TYPE ST_EL3446_MUX_ULINT :
STRUCT
    nSelector : UINT := E_EL3446_Phase.Error_INDEX_Not_Valid;
    nValueRef : POINTER TO ULINT;
END_STRUCT
END_TYPE

(* stored: Version 1.1.0.1, ProductVersion 3.1.4024.12
   DUT ST_EL3446_MUX_ULINT: Id {96135ce8-a2c3-425e-8e96-aa2e7ed6d1de} *)
